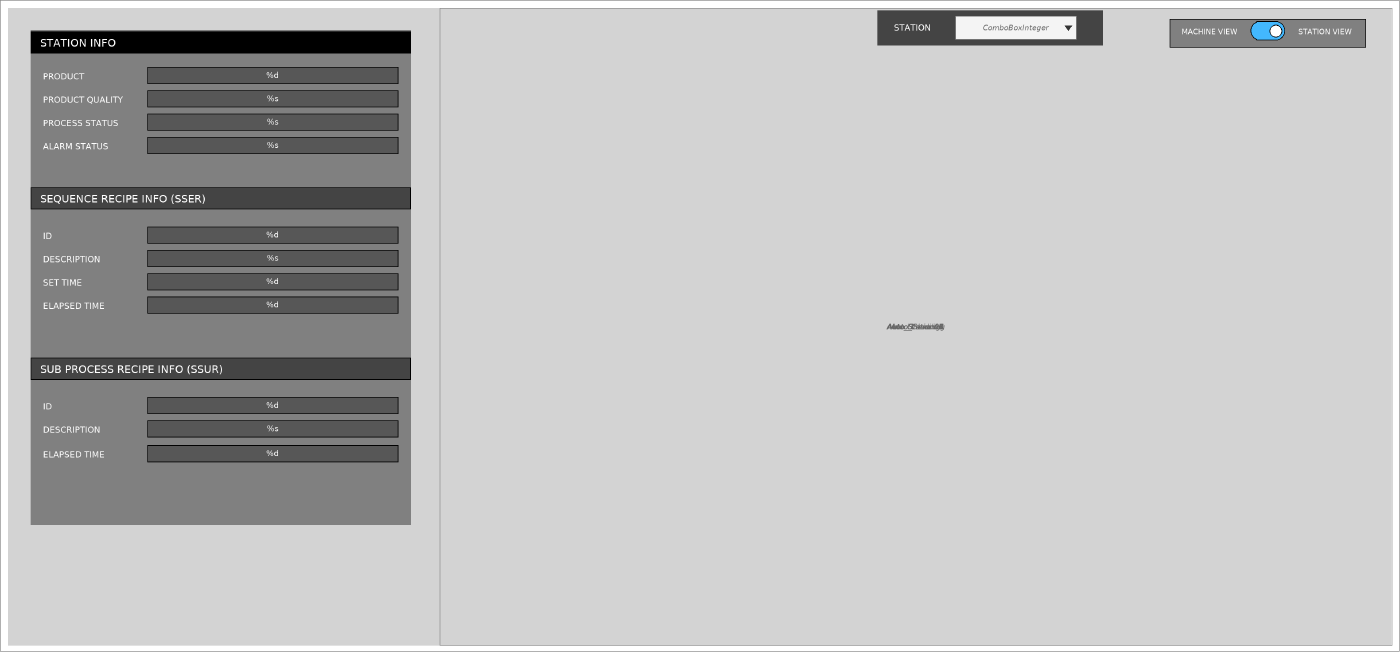
VISUALIZATION Auto_AllStation  // 1920x895
    Rectangle (0,0 1920x895)
    Rectangle (11,11 1896x875)
    Rectangle (42,41 521x679)
    Group (42,43 521x30)
        Rectangle (0,0 521x30)
        Label (10,8 150x16), "STATION INFO"
    Label (56,129 150x16), "PRODUCT QUALITY"
    Rectangle (202,124 344x23), "%s", text variable: DSStnBasketInfo[iAutoStnInfoPageNo].sProductQuality
    Label (56,161 150x16), "PROCESS STATUS"
    Rectangle (202,156 344x23), "%s", text variable: ARsStnProcessStatus[iAutoStnInfoPageNo]
    Label (56,193 150x16), "ALARM STATUS"
    Rectangle (202,188 344x23), "%s", text variable: DSHmiStationDisplayInfo[iAutoStnInfoPageNo].sErrorMessage
    Label (56,412 150x16), "ELAPSED TIME"
    Rectangle (202,407 344x23), "%d", text variable: ARDsStnSeqProcessCtrl[iAutoStnInfoPageNo].Out_iTotalProcessTimeEV
    Label (56,316 150x16), "ID"
    Rectangle (202,311 344x23), "%d", text variable: DSStnBasketInfo[iAutoStnInfoPageNo].iStationSeqenceRecipeNo
    Label (56,348 150x16), "DESCRIPTION"
    Rectangle (202,343 344x23), "%s", text variable: DSHmiStationDisplayInfo[iAutoStnInfoPageNo].sStationSequenceRecipeDescription
    Label (56,380 150x16), "SET TIME"
    Rectangle (202,375 344x23), "%d", text variable: ARDsStnMinMaxEffTimeDisplay[iAutoStnInfoPageNo].iEffTime
    Rectangle (42,257 521x30)
    Label (52,265 496x16), "SEQUENCE RECIPE INFO (SSER)"
    Label (56,616 150x16), "ELAPSED TIME"
    Rectangle (202,611 344x23), "%d", text variable: ARDsStnSeqProcessCtrl[iAutoStnInfoPageNo].Out_iComConProcessTimeEV
    Label (56,550 150x16), "ID"
    Rectangle (202,545 344x23), "%d", text variable: DSStnBasketInfo[iAutoStnInfoPageNo].iProductRecipeStepNo
    Label (56,582 150x16), "DESCRIPTION"
    Rectangle (202,577 344x23), "%s", text variable: DSHmiStationDisplayInfo[iAutoStnInfoPageNo].sStationSubDescription
    Rectangle (42,491 521x30)
    Label (52,499 492x16), "SUB PROCESS RECIPE INFO (SSUR)"
    Rectangle (202,92 344x23), "%d", text variable: DSStnBasketInfo[iAutoStnInfoPageNo].iProductRecipeNo
    Label (56,97 150x16), "PRODUCT"
    Group (603,11 1306x875)
        Frame (0,0 1306x875), invisible if: iAutoStnInfoPageNo <> 2
            shows Auto_Station02()
        Frame (0,0 1306x875), invisible if: iAutoStnInfoPageNo <> 1
            shows Auto_Station01()
        Frame (0,0 1306x875), invisible if: iAutoStnInfoPageNo<> 3
            shows Auto_Station03()
        Frame (0,0 1306x875), invisible if: iAutoStnInfoPageNo <> 4
            shows Auto_Station04()
        Frame (0,0 1306x875), invisible if: iAutoStnInfoPageNo <> 5
            shows Auto_Station05()
        Frame (0,0 1306x875), invisible if: iAutoStnInfoPageNo <> 6
            shows Auto_Station06()
        Frame (0,0 1306x875), invisible if: iAutoStnInfoPageNo <> 7
            shows Auto_Loading()
        Frame (0,0 1306x875), invisible if: iAutoStnInfoPageNo<> 8
            shows Auto_Unloading()
        Frame (0,0 1306x875), invisible if: iAutoStnInfoPageNo<> 9
            shows Auto_General()
    RoundedRectangle (1604,26 269x39)
    Label (1605,23 108x41), "MACHINE VIEW"
    Label (1765,23 105x41), "STATION VIEW"
    Group (1715,29 47x26)
        OnMouseClick: toggle HMI_Ctrl.AutoStationViewEnable
        Group (0,0 47x26)
            Ellipse (0,0 26x26)
            Ellipse (21,0 26x26)
            RoundedRectangle (8,0 29x26)
        Ellipse (1,1 24x24)
        Ellipse (23,1 23x24)
        RoundedRectangle (9,1 28x24)
        Ellipse (26,5 17x17)
    Group (1203,14 288x48)
        RoundedRectangle (0,0 309x48)
        Label (20,12 79x24), "STATION"
    ComboBoxInteger (1310,22 166x32), variable: iAutoStnInfoPageNo, invisible if: NOT HMI_Ctrl.AutoStationViewEnable, text list: 'TextList_SettingPage'
END_VISUALIZATION

(* stored: Version 1.1.0.1, ProductVersion 3.1.4024.12
   Visu Auto_AllStation: Id {4e538fc2-671e-4b67-85fb-afc1b461d6a0} *)
